KUKA KRL program: PULLTEST.src, PULLTEST.dat

--- PULLTEST.src ---
&ACCESS RVP
&REL 10
&PARAM TEMPLATE = C:\KRC\Roboter\Template\vorgabe
&PARAM EDITMASK = *
DEF PULLTEST( )
INT X
DECL BOOL TEMP, SEMP, HEMP
DECL FRAME PT1, PT2
DECL CHAR DIRECTION
DECL INT SIGN
DECL CHAR FORCE[13]
DECL REAL FZ,STIFFNESS

;FOLD INI
  ;FOLD BASISTECH INI
    GLOBAL INTERRUPT DECL 3 WHEN $STOPMESS==TRUE DO IR_STOPM ( )
    INTERRUPT ON 3
    BAS (#INITMOV,0 )
  ;ENDFOLD (BASISTECH INI)
  ;FOLD USER INI
    ;Make your modifications here
  ;ENDFOLD (USER INI)
;ENDFOLD (INI)

$ADVANCE=3

$STIFFNESS.STRATEGY=10
$STIFFNESS.COMMIT=TRUE
$ORI_TYPE=#CONSTANT
$TOOL=TOOL_DATA[4]
$VEL.CP=1.0
$VEL.ORI1=100
$VEL.ORI2=100
$ACC.CP=1.0
$ACC.ORI1=100
$ACC.ORI2=100
FOR X=1 TO 6
$ACC_AXIS[X]=100
$VEL_AXIS[X]=100
ENDFOR

;CHANGE THIS EACH TIME
;SIGN=1 IS POSITIVE
;SIGN=-1 IS NEGATIVE
DIRECTION="V"
SIGN=-1
STIFFNESS=10
$OV_PRO=40


;FOLD PTP P3 Vel=100 % PDAT3 Tool[4]:Pneumatic_gripper Base[0];%{PE}%R 5.6.11,%MKUKATPBASIS,%CMOVE,%VPTP,%P 1:PTP, 2:P3, 3:, 5:100, 7:PDAT3
$BWDSTART=FALSE
PDAT_ACT=PPDAT3
FDAT_ACT=FP3
BAS(#PTP_PARAMS,100)
PTP XP3
;ENDFOLD


;PT1= GETPOINT(DIRECTION,SIGN)
;PTP PT1

;TEMP=TRIG()

SEMP=SETSTIFF(DIRECTION,STIFFNESS)

;HEMP=SETFORCE(DIRECTION,FZ)


;LIN_REL PT2

;WAIT SEC 5

;$STIFFNESS.STRATEGY=10
;$STIFFNESS.COMMIT=TRUE
;$OV_PRO=40

;LIN_REL {Z 30}






END

--- PULLTEST.dat ---
&ACCESS RVP
&REL 10
&PARAM TEMPLATE = C:\KRC\Roboter\Template\vorgabe
&PARAM EDITMASK = *
DEFDAT  PULLTEST
;FOLD EXTERNAL DECLARATIONS;%{PE}%MKUKATPBASIS,%CEXT,%VCOMMON,%P
;FOLD BASISTECH EXT;%{PE}%MKUKATPBASIS,%CEXT,%VEXT,%P
EXT  BAS (BAS_COMMAND  :IN,REAL  :IN )
DECL INT SUCCESS
;ENDFOLD (BASISTECH EXT)
;FOLD USER EXT;%{E}%MKUKATPUSER,%CEXT,%VEXT,%P
;Make here your modifications

;ENDFOLD (USER EXT)
;ENDFOLD (EXTERNAL DECLARATIONS)
DECL BASIS_SUGG_T LAST_BASIS={POINT1[] "P3                      ",POINT2[] "P3                      ",CP_PARAMS[] "CPDAT0                  ",PTP_PARAMS[] "PDAT3                   ",CONT[] "                        ",CP_VEL[] "2.0                     ",PTP_VEL[] "100                     ",SYNC_PARAMS[] "SYNCDAT                 ",SPL_NAME[] "S0                      "}
DECL E6POS XP1={X 12.30126,Y -591.60022,Z 156.144394,A 1.17926598,B -0.00117073196,C -179.9776,S 1,T 36,E1 -0.0129604302,E2 0.0,E3 0.0,E4 0.0,E5 0.0,E6 0.0}
DECL FDAT FP1={TOOL_NO 5,BASE_NO 0,IPO_FRAME #BASE,POINT2[] " ",TQ_STATE FALSE}
DECL PDAT PPDAT1={VEL 100.0,ACC 100.0,APO_DIST 100.0,APO_MODE #CPTP}
DECL INT LAST_XP_POINT=1
DECL E6POS XP2={X 12.30126,Y -591.60022,Z 156.144394,A 1.17926598,B -0.00117073196,C -179.9776,S 1,T 36,E1 -0.0129604302,E2 0.0,E3 0.0,E4 0.0,E5 0.0,E6 0.0}
DECL FDAT FP2={TOOL_NO 5,BASE_NO 0,IPO_FRAME #BASE,POINT2[] " ",TQ_STATE FALSE}
DECL PDAT PPDAT2={VEL 100.0,ACC 100.0,APO_DIST 100.0,APO_MODE #CPTP}
DECL E6POS XP3={X 32.4354401,Y -634.169128,Z 349.833099,A 87.7409363,B 27.0057297,C 178.216202,S 6,T 49,E1 -24.0416603,E2 0.0,E3 0.0,E4 0.0,E5 0.0,E6 0.0}
DECL FDAT FP3={TOOL_NO 4,BASE_NO 0,IPO_FRAME #BASE,POINT2[] " ",TQ_STATE FALSE}
DECL PDAT PPDAT3={VEL 100.0,ACC 100.0,APO_DIST 100.0,APO_MODE #CPTP}
ENDDAT
